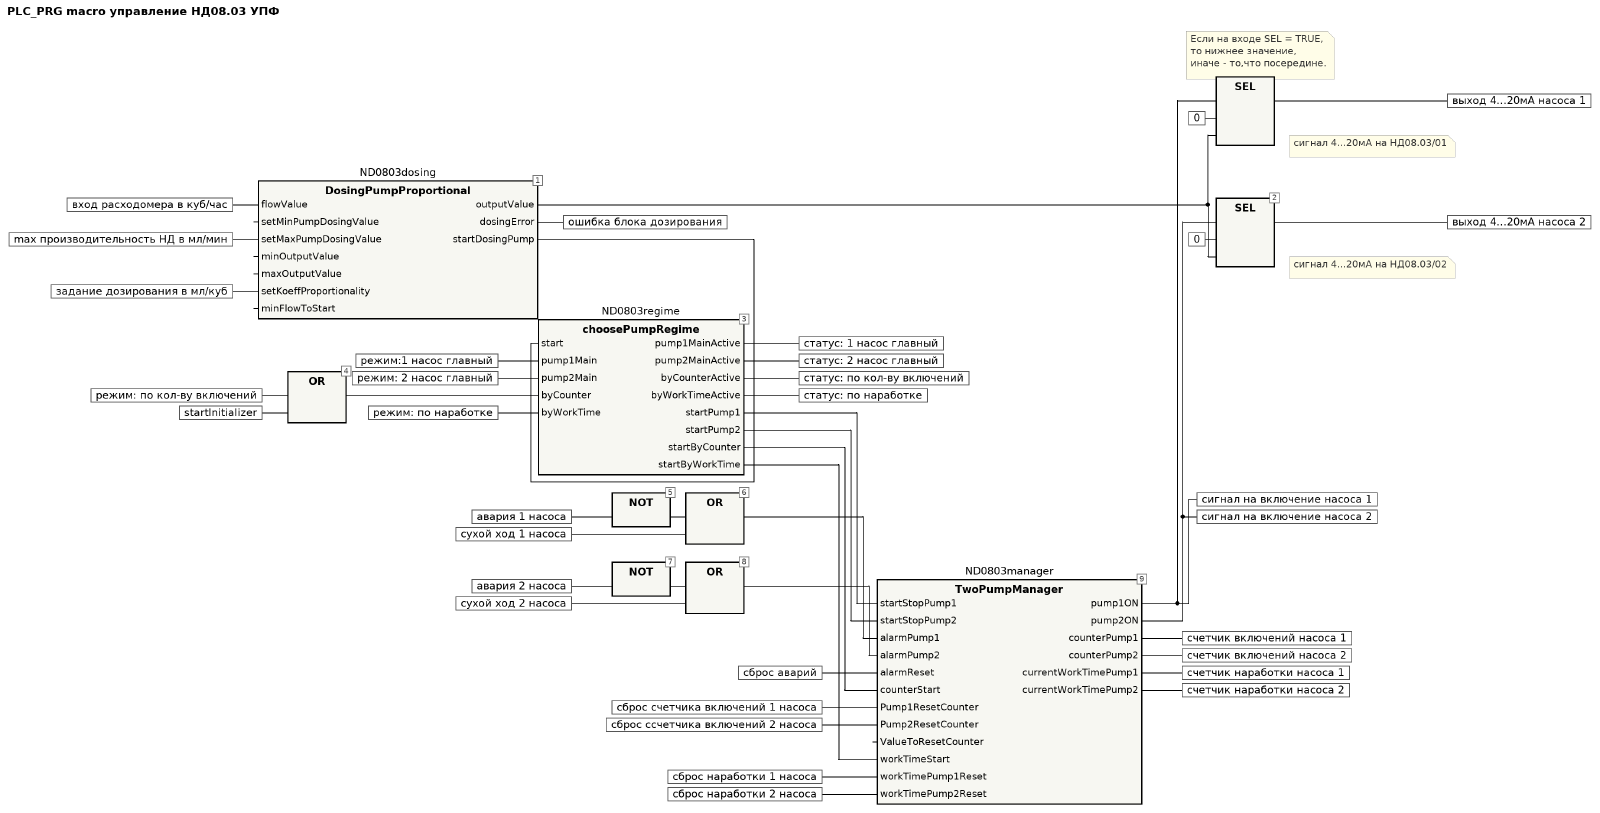
[picture p24: PLC_PRG macro управление НД08.03 УПФ (CFC)]
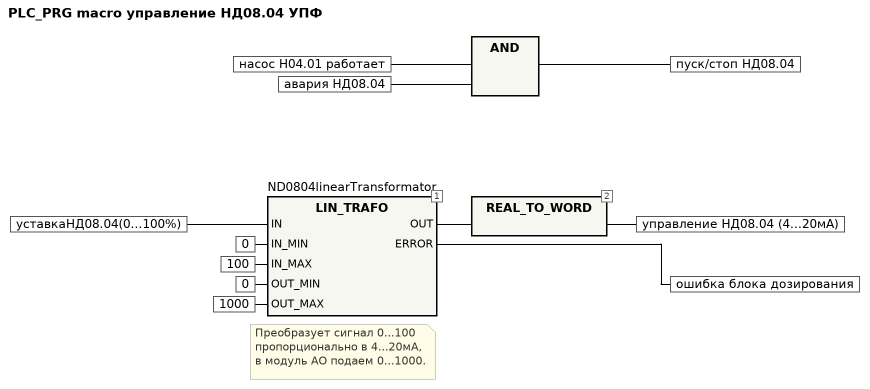
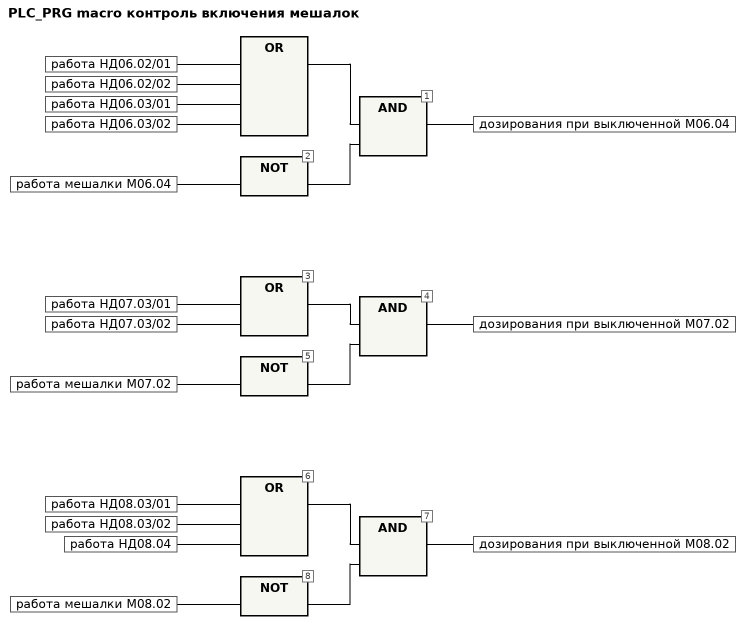
[picture p26: PLC_PRG macro контроль включения мешалок (CFC)]
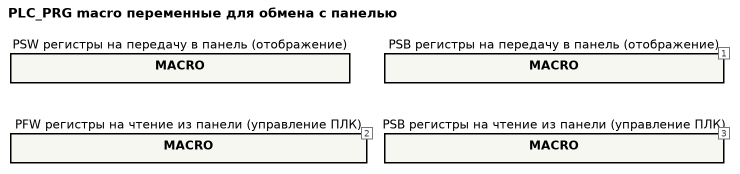
[picture p27: PLC_PRG macro переменные для обмена с панелью (CFC)]
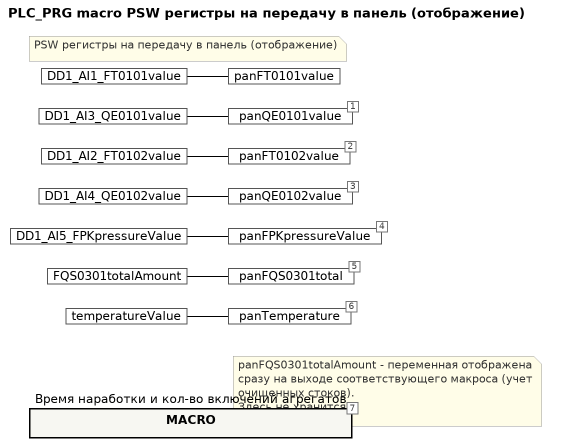
[picture p28: PLC_PRG macro PSW регистры на передачу в панель (отображение) (CFC)]
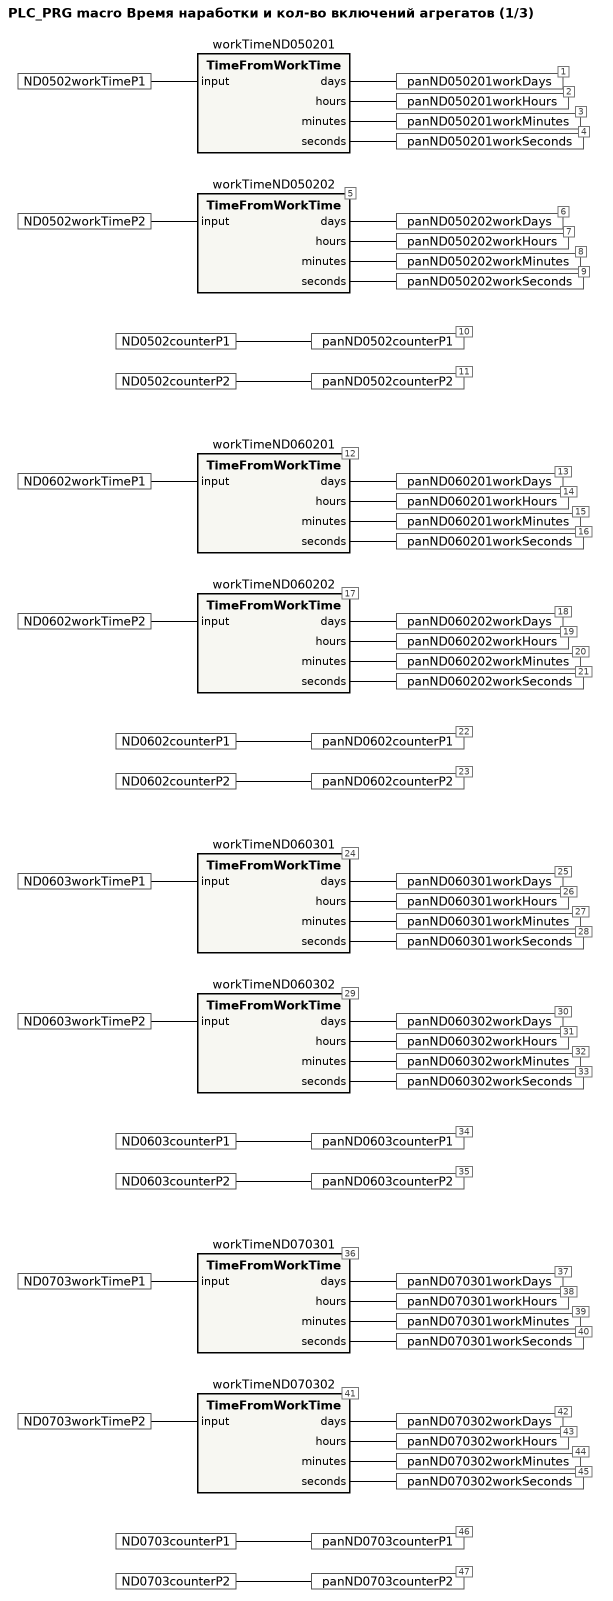
[picture p29: PLC_PRG macro Время наработки и кол-во включений агрегатов (CFC)]
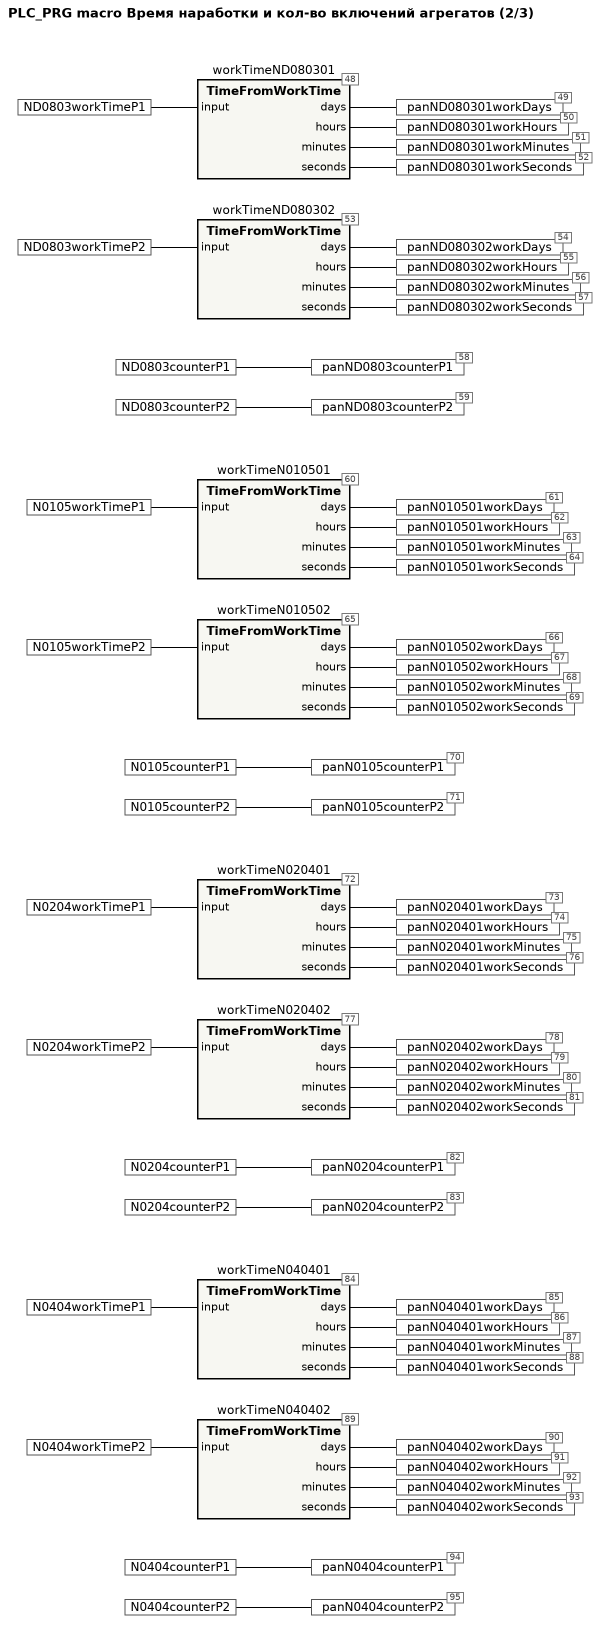
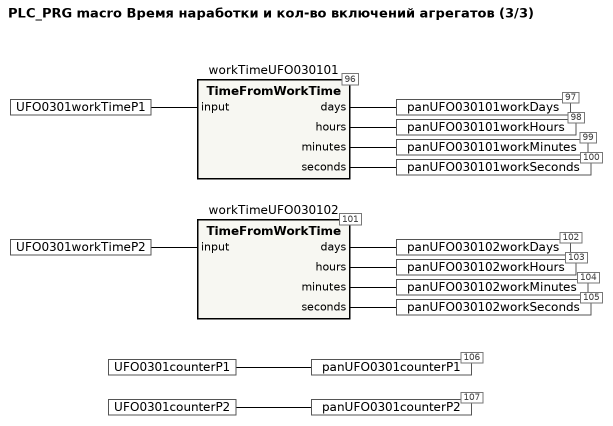
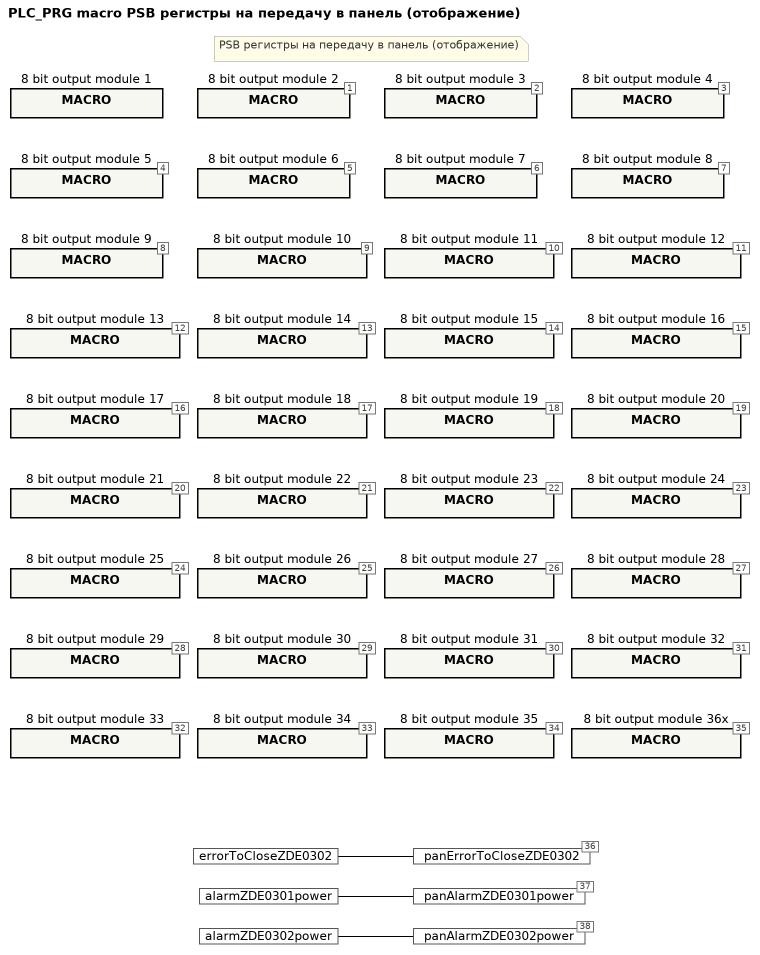
[picture p32: PLC_PRG macro PSB регистры на передачу в панель (отображение) (CFC)]
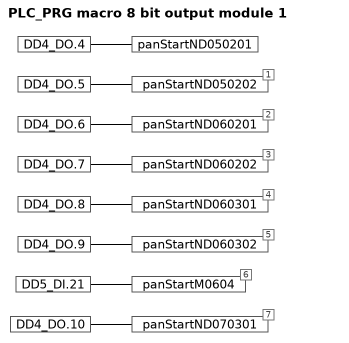
[picture p33: PLC_PRG macro 8 bit output module 1 (CFC)]
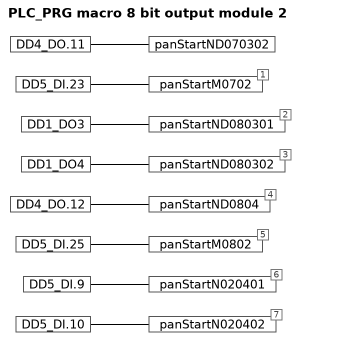
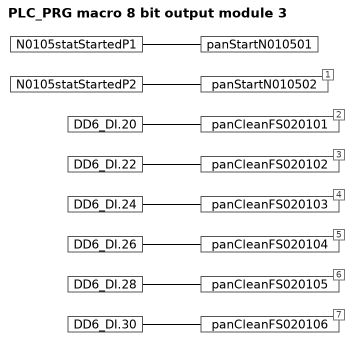
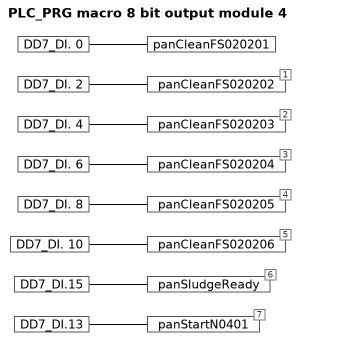
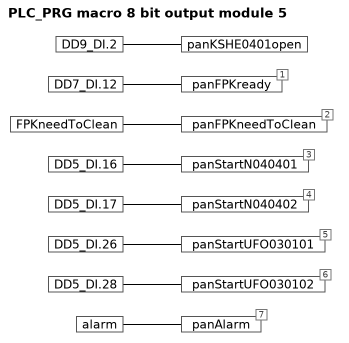
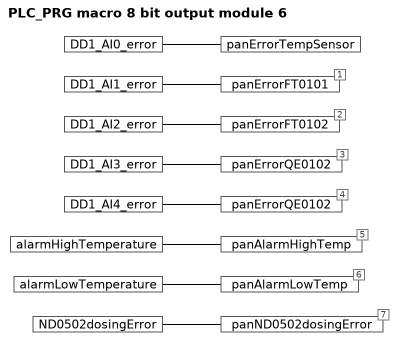
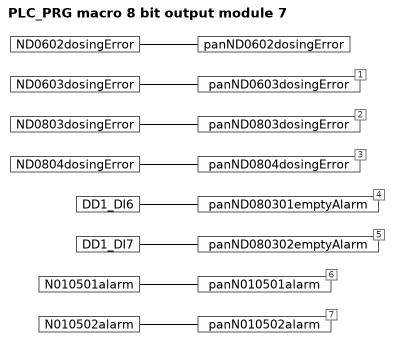
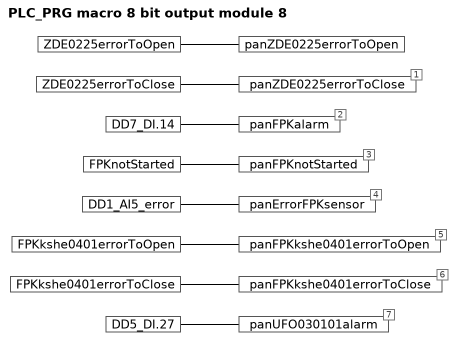
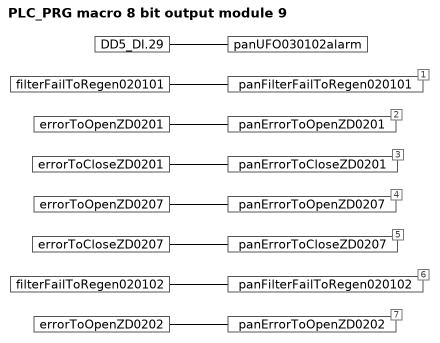
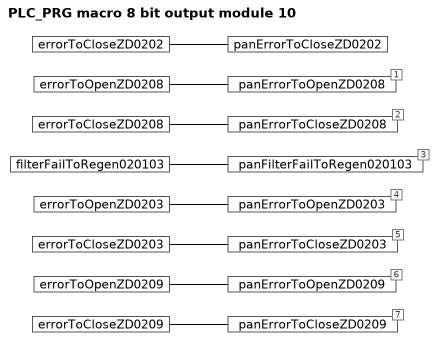
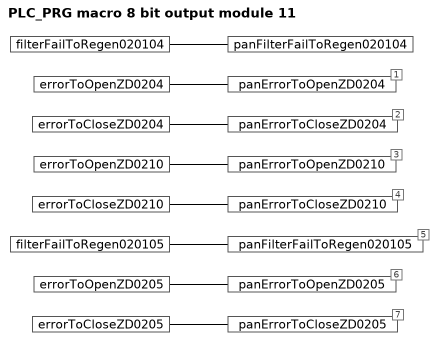
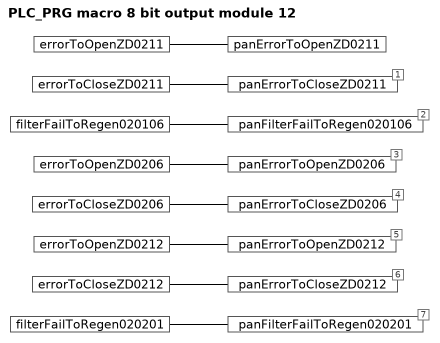
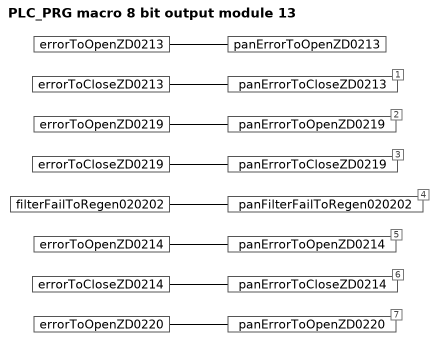
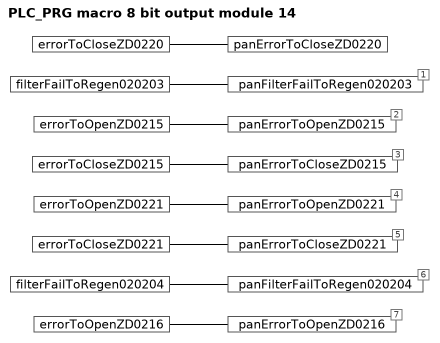
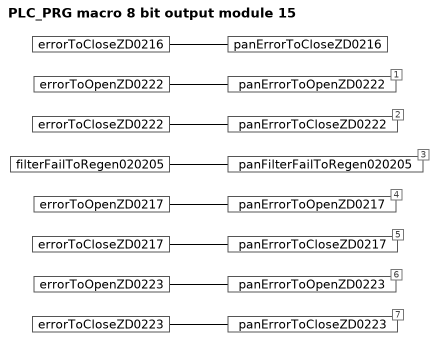
